# EPICS autosave request: iocs/meascomp/usb-2408-ioc/auto_settings.req
# Settings restored at the next start of usb-2408-ioc.
# Ported from upstream USB2408_settings.req and the per-template
# measComp*_settings.req files it includes, minus the records this port does
# not have (Ao SyncMaster: the USB-2408-2AO rejects AO_CFG_SYNC_MODE).
#
# Macros: P (record prefix)

$(P)PollSleepMS

$(P)Bd1
$(P)Bd2
$(P)Bd3
$(P)Bd4
$(P)Bd5
$(P)Bd6
$(P)Bd7
$(P)Bd8

$(P)AiMode

$(P)Ai1Range
$(P)Ai1Type
$(P)Ai1Rate
$(P)Ai1.LOPR
$(P)Ai1.HOPR
$(P)Ai1.EGUF
$(P)Ai1.EGUL
$(P)Ai1.PREC
$(P)Ai1.SCAN
$(P)Ai2Range
$(P)Ai2Type
$(P)Ai2Rate
$(P)Ai2.LOPR
$(P)Ai2.HOPR
$(P)Ai2.EGUF
$(P)Ai2.EGUL
$(P)Ai2.PREC
$(P)Ai2.SCAN
$(P)Ai3Range
$(P)Ai3Type
$(P)Ai3Rate
$(P)Ai3.LOPR
$(P)Ai3.HOPR
$(P)Ai3.EGUF
$(P)Ai3.EGUL
$(P)Ai3.PREC
$(P)Ai3.SCAN
$(P)Ai4Range
$(P)Ai4Type
$(P)Ai4Rate
$(P)Ai4.LOPR
$(P)Ai4.HOPR
$(P)Ai4.EGUF
$(P)Ai4.EGUL
$(P)Ai4.PREC
$(P)Ai4.SCAN
$(P)Ai5Range
$(P)Ai5Type
$(P)Ai5Rate
$(P)Ai5.LOPR
$(P)Ai5.HOPR
$(P)Ai5.EGUF
$(P)Ai5.EGUL
$(P)Ai5.PREC
$(P)Ai5.SCAN
$(P)Ai6Range
$(P)Ai6Type
$(P)Ai6Rate
$(P)Ai6.LOPR
$(P)Ai6.HOPR
$(P)Ai6.EGUF
$(P)Ai6.EGUL
$(P)Ai6.PREC
$(P)Ai6.SCAN
$(P)Ai7Range
$(P)Ai7Type
$(P)Ai7Rate
$(P)Ai7.LOPR
$(P)Ai7.HOPR
$(P)Ai7.EGUF
$(P)Ai7.EGUL
$(P)Ai7.PREC
$(P)Ai7.SCAN
$(P)Ai8Range
$(P)Ai8Type
$(P)Ai8Rate
$(P)Ai8.LOPR
$(P)Ai8.HOPR
$(P)Ai8.EGUF
$(P)Ai8.EGUL
$(P)Ai8.PREC
$(P)Ai8.SCAN

$(P)Ti1Scale
$(P)Ti1TCType
$(P)Ti1OpenTCDetect
$(P)Ti1Filter
$(P)Ti1.LOPR
$(P)Ti1.HOPR
$(P)Ti1.PREC
$(P)Ti1.SCAN
$(P)Ti2Scale
$(P)Ti2TCType
$(P)Ti2OpenTCDetect
$(P)Ti2Filter
$(P)Ti2.LOPR
$(P)Ti2.HOPR
$(P)Ti2.PREC
$(P)Ti2.SCAN
$(P)Ti3Scale
$(P)Ti3TCType
$(P)Ti3OpenTCDetect
$(P)Ti3Filter
$(P)Ti3.LOPR
$(P)Ti3.HOPR
$(P)Ti3.PREC
$(P)Ti3.SCAN
$(P)Ti4Scale
$(P)Ti4TCType
$(P)Ti4OpenTCDetect
$(P)Ti4Filter
$(P)Ti4.LOPR
$(P)Ti4.HOPR
$(P)Ti4.PREC
$(P)Ti4.SCAN
$(P)Ti5Scale
$(P)Ti5TCType
$(P)Ti5OpenTCDetect
$(P)Ti5Filter
$(P)Ti5.LOPR
$(P)Ti5.HOPR
$(P)Ti5.PREC
$(P)Ti5.SCAN
$(P)Ti6Scale
$(P)Ti6TCType
$(P)Ti6OpenTCDetect
$(P)Ti6Filter
$(P)Ti6.LOPR
$(P)Ti6.HOPR
$(P)Ti6.PREC
$(P)Ti6.SCAN
$(P)Ti7Scale
$(P)Ti7TCType
$(P)Ti7OpenTCDetect
$(P)Ti7Filter
$(P)Ti7.LOPR
$(P)Ti7.HOPR
$(P)Ti7.PREC
$(P)Ti7.SCAN
$(P)Ti8Scale
$(P)Ti8TCType
$(P)Ti8OpenTCDetect
$(P)Ti8Filter
$(P)Ti8.LOPR
$(P)Ti8.HOPR
$(P)Ti8.PREC
$(P)Ti8.SCAN

$(P)Ao1Range
$(P)Ao1TweakVal
$(P)Ao1SyncEnable
$(P)Ao1Pulse
$(P)Ao1.DRVL
$(P)Ao1.DRVH
$(P)Ao1.LOPR
$(P)Ao1.HOPR
$(P)Ao1.EGUF
$(P)Ao1.EGUL
$(P)Ao1.PREC
$(P)Ao1Return.DRVL
$(P)Ao1Return.DRVH
$(P)Ao1Return.LOPR
$(P)Ao1Return.HOPR
$(P)Ao1Return.EGUF
$(P)Ao1Return.EGUL
$(P)Ao1Return.PREC
$(P)Ao2Range
$(P)Ao2TweakVal
$(P)Ao2SyncEnable
$(P)Ao2Pulse
$(P)Ao2.DRVL
$(P)Ao2.DRVH
$(P)Ao2.LOPR
$(P)Ao2.HOPR
$(P)Ao2.EGUF
$(P)Ao2.EGUL
$(P)Ao2.PREC
$(P)Ao2Return.DRVL
$(P)Ao2Return.DRVH
$(P)Ao2Return.LOPR
$(P)Ao2Return.HOPR
$(P)Ao2Return.EGUF
$(P)Ao2Return.EGUL
$(P)Ao2Return.PREC

$(P)WaveDigNumPoints
$(P)WaveDigFirstChan
$(P)WaveDigNumChans
$(P)WaveDigDwell
$(P)WaveDigExtTrigger
$(P)WaveDigExtClock
$(P)WaveDigContinuous
$(P)WaveDigAutoRestart
$(P)WaveDigRetrigger
$(P)WaveDigTriggerCount
$(P)WaveDigBurstMode
$(P)WaveDigReadWF.SCAN

$(P)WaveGenUserNumPoints
$(P)WaveGenIntNumPoints
$(P)WaveGenUserDwell
$(P)WaveGenIntDwell
$(P)WaveGenExtTrigger
$(P)WaveGenExtClock
$(P)WaveGenContinuous
$(P)WaveGenRetrigger
$(P)WaveGenTriggerCount

$(P)WaveGen1Enable
$(P)WaveGen1WaveType
$(P)WaveGen1PulseWidth
$(P)WaveGen1PulseDelay
$(P)WaveGen1Amplitude
$(P)WaveGen1Offset
$(P)WaveGen2Enable
$(P)WaveGen2WaveType
$(P)WaveGen2PulseWidth
$(P)WaveGen2PulseDelay
$(P)WaveGen2Amplitude
$(P)WaveGen2Offset
